{attribute 'no_explicit_call' := 'This is a CLASS and should be accessed using methods or properties'}
FUNCTION_BLOCK tempSensor_PT1000 EXTENDS tempSensor
(*~
<docu>
	<summary>
			Implementation of a PT1000 Temperature sensor class based on the base class tempSensor

			Usage:
			degreesC / degreesF return the Celcius / Fahrenheit value determined by the appropriate formula 		
	</summary>				
</docu>	
~*)

(*  
	Principally a CLASS should be accessed using methods or properties
	Good practice is not put code here, or call the class directly 
	Or maybe just a call to a method calling the cyclic code 
*)

PROPERTY tempDegreesC : REAL
GET
tempDegreesC := TEMP_PT(
			Res	:= TO_REAL(rawValue), 
			R0	:= 1000.0
			);
END_GET
END_PROPERTY

END_FUNCTION_BLOCK

(* stored: Version 1.1.0.1, ProductVersion 3.1.4024.12
   POU tempSensor_PT1000: Id {c0c66743-b10d-45bf-ad67-6e8c1b0f5e19}, SpecialFunc None
   Property tempDegreesC: Id {bb4b1eaa-4186-48ef-9f66-c5c9e653d108}
   Get Get: Id {2725969b-6912-427b-bca3-12aff0d2d250} *)
